Staubli VAL3: moveTest.pgx

public program moveTest()
  local jointRx l_jJointRx_Me
  local jointRx l_jJointRx_Bro
begin

  l_jJointRx_Me={0,0,0,0,0,0}

  //测试机器人通讯
  while true

    movej(l_jJointRx_Me,flange,mNomSpeed)
    waitEndMove()
    delay(0.5)
    call Communication(l_jJointRx_Me,l_jJointRx_Bro)

    l_jJointRx_Me.j1=l_jJointRx_Me.j1+1
    l_jJointRx_Me.j2=l_jJointRx_Me.j2+1
    l_jJointRx_Me.j3=l_jJointRx_Me.j3+1
    l_jJointRx_Me.j4=l_jJointRx_Me.j4+1
    l_jJointRx_Me.j5=l_jJointRx_Me.j5+1
    l_jJointRx_Me.j6=l_jJointRx_Me.j6+1

  endWhile
end
